FUNCTION_BLOCK FB_Button
VAR
	sButtonName : STRING;
	bExecute : BOOL;
	ExecuteCounter : UDINT;
	_refCommand : REFERENCE TO E_Command;
	InputCommand : E_Command;
	_iLog : I_Log;
	Rtrig : R_TRIG;
END_VAR

IF bExecute THEN
	ExecuteCounter := ExecuteCounter + _TaskInfo[1].CycleTime/10000;
	IF ExecuteCounter >= 1000 THEN
		_refCommand := InputCommand;
		bExecute := FALSE;
	END_IF
ELSE
	ExecuteCounter := 0;
END_IF

Rtrig(CLK := bExecute);
IF Rtrig.Q THEN
	_iLog.AddLog(CONCAT(TO_STRING(InputCommand),' is pushed'));
END_IF

METHOD FB_init : BOOL
VAR_INPUT
	bInitRetains : BOOL; // if TRUE, the retain variables are initialized (warm start / cold start)
	bInCopyCode : BOOL;  // if TRUE, the instance afterwards gets moved into the copy code (online change)
	InputCommand : E_Command;
END_VAR
sButtonName := TO_STRING(InputCommand);
THIS^.InputCommand := InputCommand;
END_METHOD

PROPERTY iLog : I_Log
GET
iLog := _iLog;
END_GET
SET
_iLog := iLog;
END_SET
END_PROPERTY

PROPERTY refCommand : REFERENCE TO E_COMMAND
GET
refCommand REF= _refCommand;
END_GET
SET
 _refCommand REF= refCommand;
END_SET
END_PROPERTY

END_FUNCTION_BLOCK

(* stored: Version 1.1.0.1, ProductVersion 3.1.4024.12
   POU FB_Button: Id {39098658-c1cc-443a-8bd8-27357fe3de3f}, SpecialFunc None
   Method FB_init: Id {a06ebe7b-8ec2-4b35-b5cb-0e5d01f70279}
   Property iLog: Id {74ef2c1a-42c4-4dc6-8259-122ec63298da}
   Get Get: Id {7c961496-18d7-400e-8afc-dfbebabe162f}
   Set Set: Id {49e2d186-5831-4ef1-9458-8dceb3c0ffe6}
   Property refCommand: Id {0e6473e5-1846-4915-90bf-477765414c6a}
   Get Get: Id {cd70e42c-fb39-40c2-9e62-cac9dacd99c1}
   Set Set: Id {13e8ebc9-02fb-40fd-9251-62421fc736b2} *)
